REGION Network 71: Call CM Expel FWD/BWD (LBC_TwoWayActuator)
   RUNG wire#powerrail
      #instcmExpelFwdBwd(enable := wire#w1, enableManualCmds := wire#w2, parentReferenceDesignator := "Unit1.Em1.Config".em.referenceDesignator.combined, feedbackHomePos := "BA010AZCRBK01.01", feedbackWorkPos := "BA010AZCRBK01.11", interlockHomePos := "Unit1.Em1.ControlNodes".cm.interlock.expel.home, interlockWorkPos := "Unit1.Em1.ControlNodes".cm.interlock.expel.work, configuration := "Unit1.Em1.Config".cmExpelFwdBwd, moduleInterface := "Unit1.Em1.HmiInterface".cmExpelFwdBwd, controlNode := "Unit1.Em1.ControlNodes".cmExpelFwdBwd, goToHomePos => "BA010AZCRPM06.01", goToWorkPos => "BA010AZCRPM06.00")
   END_RUNG
   RUNG wire#powerrail
      I_Contact( #statUnitStatus.state.aborted )
   END_RUNG wire#w1
   RUNG wire#powerrail
      Contact( #statEnableManualCmds )
   END_RUNG wire#w2
   RUNG wire#powerrail
      Contact( #statRcEnableCmds )
   END_RUNG wire#w2
   // the same network as SCL:
   #instcmExpelFwdBwd(enable := NOT #statUnitStatus.state.aborted,   // "LBC_TwoWayActuatorCn"
                      parentReferenceDesignator := "Unit1.Em1.Config".em.referenceDesignator.combined,
                      feedbackHomePos := "BA010AZCRBK01.01",
                      feedbackWorkPos := "BA010AZCRBK01.11",
                      enableManualCmds := #statEnableManualCmds OR #statRcEnableCmds,
                      interlockHomePos := "Unit1.Em1.ControlNodes".cm.interlock.expel.home,
                      interlockWorkPos := "Unit1.Em1.ControlNodes".cm.interlock.expel.work,
                      configuration := "Unit1.Em1.Config".cmExpelFwdBwd,
                      moduleInterface := "Unit1.Em1.HmiInterface".cmExpelFwdBwd,
                      controlNode := "Unit1.Em1.ControlNodes".cmExpelFwdBwd,
                      goToHomePos => "BA010AZCRPM06.01",
                      goToWorkPos => "BA010AZCRPM06.00");
END_REGION

REGION Network 72: ******************** Control Modules (Accessories) ********************
END_REGION

REGION Network 73: Reset CMS
   RUNG wire#powerrail
      Contact( #statUnitStatus.acknowledgeActive )
      wire#w1
      Contact( "Unit1.Em1.ControlNodes".cmEpc.monitoring.error )
      Coil( "Unit1.Em1.ControlNodes".cmEpc.commands.reset )
   END_RUNG
   RUNG wire#powerrail
      Contact( #statUnitStatus.state.resetting )
   END_RUNG wire#w1
   RUNG wire#w1
      Contact( "Unit1.Em1.HmiInterface".cmBobinID.monitoring.error )
      Coil( "Unit1.Em1.HmiInterface".cmBobinID.commands.ResetReq )
   END_RUNG
   // the same network as SCL:
   #_w1 := #statUnitStatus.acknowledgeActive OR #statUnitStatus.state.resetting;
   "Unit1.Em1.ControlNodes".cmEpc.commands.reset := #_w1 AND "Unit1.Em1.ControlNodes".cmEpc.monitoring.error;
   "Unit1.Em1.HmiInterface".cmBobinID.commands.ResetReq := #_w1 AND "Unit1.Em1.HmiInterface".cmBobinID.monitoring.error;
END_REGION

REGION Network 74: Call CM EPC Commands
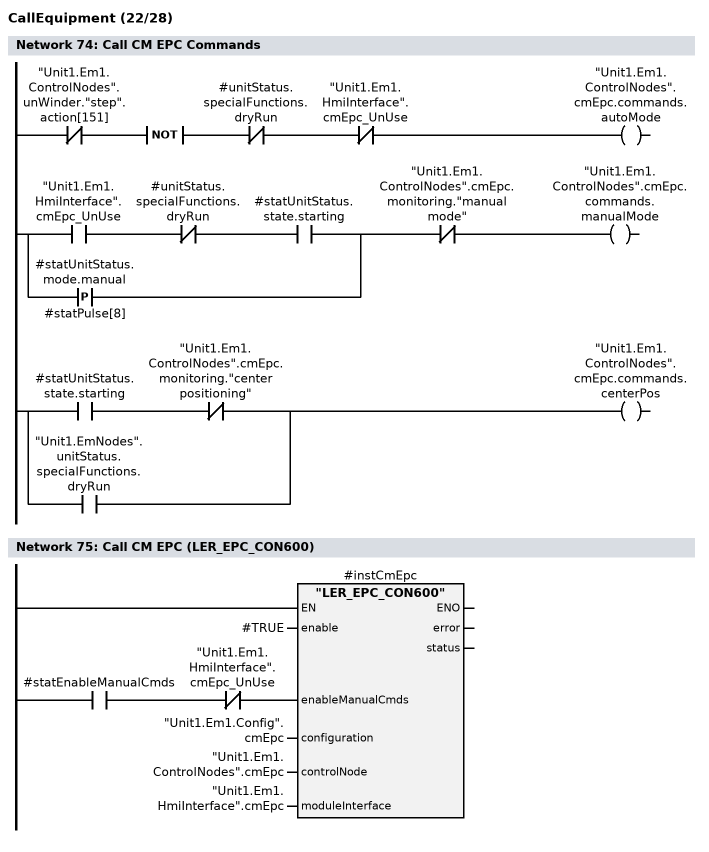
   RUNG wire#powerrail
      I_Contact( "Unit1.Em1.ControlNodes".unWinder."step".action[151] )
      Not()
      I_Contact( #unitStatus.specialFunctions.dryRun )
      I_Contact( "Unit1.Em1.HmiInterface".cmEpc_UnUse )
      Coil( "Unit1.Em1.ControlNodes".cmEpc.commands.autoMode )
   END_RUNG
   RUNG wire#powerrail
      Contact( "Unit1.Em1.HmiInterface".cmEpc_UnUse )
      I_Contact( #unitStatus.specialFunctions.dryRun )
      Contact( #statUnitStatus.state.starting )
      wire#w1
      I_Contact( "Unit1.Em1.ControlNodes".cmEpc.monitoring."manual mode" )
      Coil( "Unit1.Em1.ControlNodes".cmEpc.commands.manualMode )
   END_RUNG
   RUNG wire#powerrail
      P_Contact(operand := #statUnitStatus.mode.manual, bit := #statPulse[8])
   END_RUNG wire#w1
   RUNG wire#powerrail
      Contact( #statUnitStatus.state.starting )
      I_Contact( "Unit1.Em1.ControlNodes".cmEpc.monitoring."center positioning" )
      wire#w2
      Coil( "Unit1.Em1.ControlNodes".cmEpc.commands.centerPos )
   END_RUNG
   RUNG wire#powerrail
      Contact( "Unit1.EmNodes".unitStatus.specialFunctions.dryRun )
   END_RUNG wire#w2
   // the same network as SCL:
   "Unit1.Em1.ControlNodes".cmEpc.commands.autoMode := NOT (NOT "Unit1.Em1.ControlNodes".unWinder."step".action[151]) AND NOT #unitStatus.specialFunctions.dryRun AND NOT "Unit1.Em1.HmiInterface".cmEpc_UnUse;
   #_w1 := #statUnitStatus.mode.manual AND NOT #statPulse[8];   // rising edge of #statUnitStatus.mode.manual
   #statPulse[8] := #statUnitStatus.mode.manual;
   "Unit1.Em1.ControlNodes".cmEpc.commands.manualMode := (("Unit1.Em1.HmiInterface".cmEpc_UnUse AND NOT #unitStatus.specialFunctions.dryRun AND #statUnitStatus.state.starting) OR #_w1) AND NOT "Unit1.Em1.ControlNodes".cmEpc.monitoring."manual mode";
   "Unit1.Em1.ControlNodes".cmEpc.commands.centerPos := (#statUnitStatus.state.starting AND NOT "Unit1.Em1.ControlNodes".cmEpc.monitoring."center positioning") OR "Unit1.EmNodes".unitStatus.specialFunctions.dryRun;
END_REGION

REGION Network 75: Call CM EPC (LER_EPC_CON600)
   RUNG wire#powerrail
      #instCmEpc(enableManualCmds := wire#w1, enable := #TRUE, configuration := "Unit1.Em1.Config".cmEpc, controlNode := "Unit1.Em1.ControlNodes".cmEpc, moduleInterface := "Unit1.Em1.HmiInterface".cmEpc, error =>, status =>)
   END_RUNG
   RUNG wire#powerrail
      Contact( #statEnableManualCmds )
      I_Contact( "Unit1.Em1.HmiInterface".cmEpc_UnUse )
   END_RUNG wire#w1
   // the same network as SCL:
   #instCmEpc(enable := #TRUE,   // "LER_EPC_CON600"
              enableManualCmds := #statEnableManualCmds AND NOT "Unit1.Em1.HmiInterface".cmEpc_UnUse,
              configuration := "Unit1.Em1.Config".cmEpc,
              controlNode := "Unit1.Em1.ControlNodes".cmEpc,
              moduleInterface := "Unit1.Em1.HmiInterface".cmEpc);
END_REGION

REGION Network 76: ******************** Feedback to Unit ********************
END_REGION

REGION Network 77: Determine StateComplete (SC) in Mode Production
   // Conditions for the Equipment Modules "stateComplete" feedback to the unit. This feedback is given when the task in for the respective state is complete.
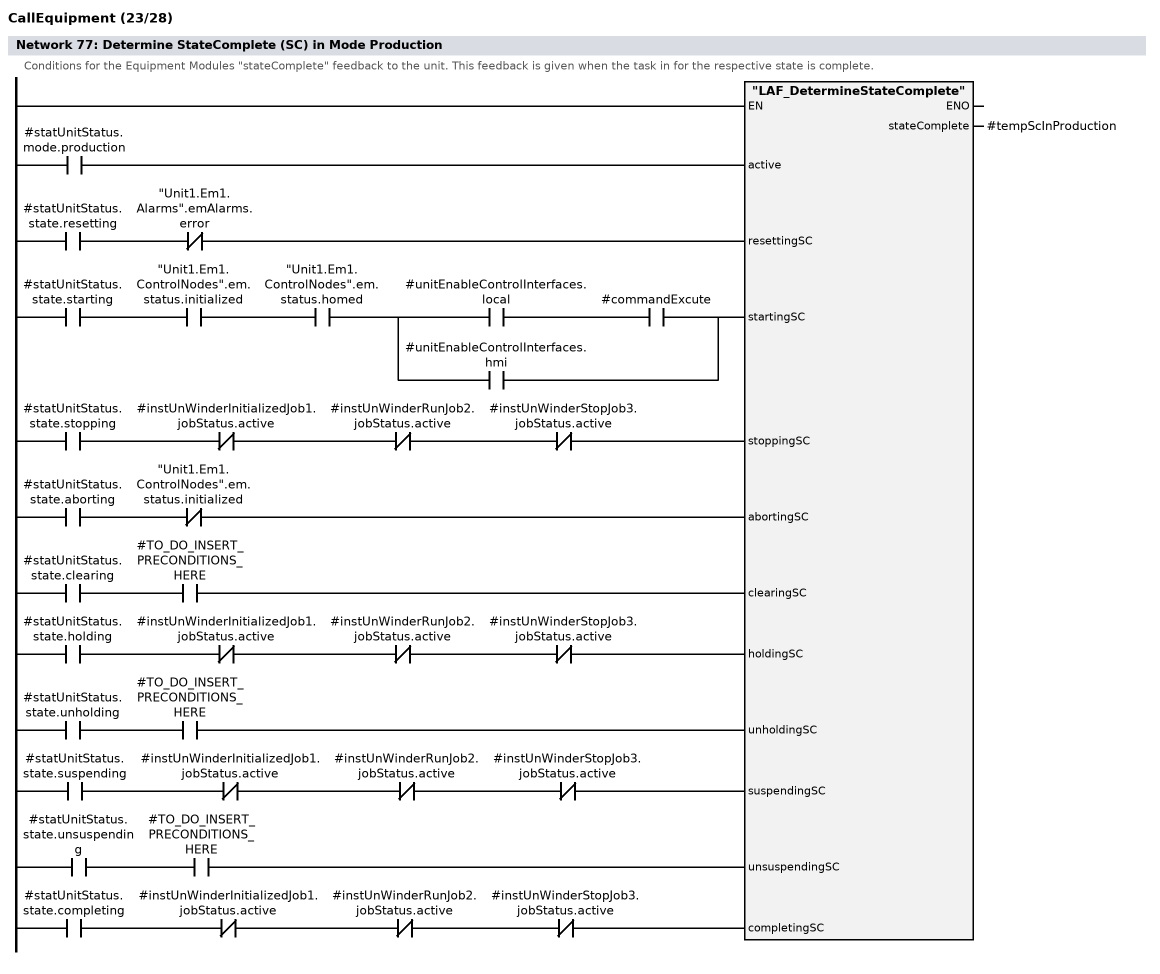
   RUNG wire#powerrail
      "LAF_DetermineStateComplete"(active := wire#w1, resettingSC := wire#w2, startingSC := wire#w4, stoppingSC := wire#w5, abortingSC := wire#w6, clearingSC := wire#w7, holdingSC := wire#w8, unholdingSC := wire#w9, suspendingSC := wire#w10, unsuspendingSC := wire#w11, completingSC := wire#w12, stateComplete => #tempScInProduction)
   END_RUNG
   RUNG wire#powerrail
      Contact( #statUnitStatus.mode.production )
   END_RUNG wire#w1
   RUNG wire#powerrail
      Contact( #statUnitStatus.state.resetting )
      I_Contact( "Unit1.Em1.Alarms".emAlarms.error )
   END_RUNG wire#w2
   RUNG wire#powerrail
      Contact( #statUnitStatus.state.starting )
      Contact( "Unit1.Em1.ControlNodes".em.status.initialized )
      Contact( "Unit1.Em1.ControlNodes".em.status.homed )
      wire#w3
      Contact( #unitEnableControlInterfaces.local )
      Contact( #commandExcute )
   END_RUNG wire#w4
   RUNG wire#w3
      Contact( #unitEnableControlInterfaces.hmi )
   END_RUNG wire#w4
   RUNG wire#powerrail
      Contact( #statUnitStatus.state.stopping )
      I_Contact( #instUnWinderInitializedJob1.jobStatus.active )
      I_Contact( #instUnWinderRunJob2.jobStatus.active )
      I_Contact( #instUnWinderStopJob3.jobStatus.active )
   END_RUNG wire#w5
   RUNG wire#powerrail
      Contact( #statUnitStatus.state.aborting )
      I_Contact( "Unit1.Em1.ControlNodes".em.status.initialized )
   END_RUNG wire#w6
   RUNG wire#powerrail
      Contact( #statUnitStatus.state.clearing )
      Contact( #TO_DO_INSERT_PRECONDITIONS_HERE )
   END_RUNG wire#w7
   RUNG wire#powerrail
      Contact( #statUnitStatus.state.holding )
      I_Contact( #instUnWinderInitializedJob1.jobStatus.active )
      I_Contact( #instUnWinderRunJob2.jobStatus.active )
      I_Contact( #instUnWinderStopJob3.jobStatus.active )
   END_RUNG wire#w8
   RUNG wire#powerrail
      Contact( #statUnitStatus.state.unholding )
      Contact( #TO_DO_INSERT_PRECONDITIONS_HERE )
   END_RUNG wire#w9
   RUNG wire#powerrail
      Contact( #statUnitStatus.state.suspending )
      I_Contact( #instUnWinderInitializedJob1.jobStatus.active )
      I_Contact( #instUnWinderRunJob2.jobStatus.active )
      I_Contact( #instUnWinderStopJob3.jobStatus.active )
   END_RUNG wire#w10
   RUNG wire#powerrail
      Contact( #statUnitStatus.state.unsuspending )
      Contact( #TO_DO_INSERT_PRECONDITIONS_HERE )
   END_RUNG wire#w11
   RUNG wire#powerrail
      Contact( #statUnitStatus.state.completing )
      I_Contact( #instUnWinderInitializedJob1.jobStatus.active )
      I_Contact( #instUnWinderRunJob2.jobStatus.active )
      I_Contact( #instUnWinderStopJob3.jobStatus.active )
   END_RUNG wire#w12
   // the same network as SCL:
   "LAF_DetermineStateComplete"(active := #statUnitStatus.mode.production,
                           resettingSC := #statUnitStatus.state.resetting AND NOT "Unit1.Em1.Alarms".emAlarms.error,
                           startingSC := #statUnitStatus.state.starting AND "Unit1.Em1.ControlNodes".em.status.initialized AND "Unit1.Em1.ControlNodes".em.status.homed AND ((#unitEnableControlInterfaces.local AND #commandExcute) OR #unitEnableControlInterfaces.hmi),
                           stoppingSC := #statUnitStatus.state.stopping AND NOT #instUnWinderInitializedJob1.jobStatus.active AND NOT #instUnWinderRunJob2.jobStatus.active AND NOT #instUnWinderStopJob3.jobStatus.active,
                           abortingSC := #statUnitStatus.state.aborting AND NOT "Unit1.Em1.ControlNodes".em.status.initialized,
                           clearingSC := #statUnitStatus.state.clearing AND #TO_DO_INSERT_PRECONDITIONS_HERE,
                           holdingSC := #statUnitStatus.state.holding AND NOT #instUnWinderInitializedJob1.jobStatus.active AND NOT #instUnWinderRunJob2.jobStatus.active AND NOT #instUnWinderStopJob3.jobStatus.active,
                           unholdingSC := #statUnitStatus.state.unholding AND #TO_DO_INSERT_PRECONDITIONS_HERE,
                           suspendingSC := #statUnitStatus.state.suspending AND NOT #instUnWinderInitializedJob1.jobStatus.active AND NOT #instUnWinderRunJob2.jobStatus.active AND NOT #instUnWinderStopJob3.jobStatus.active,
                           unsuspendingSC := #statUnitStatus.state.unsuspending AND #TO_DO_INSERT_PRECONDITIONS_HERE,
                           completingSC := #statUnitStatus.state.completing AND NOT #instUnWinderInitializedJob1.jobStatus.active AND NOT #instUnWinderRunJob2.jobStatus.active AND NOT #instUnWinderStopJob3.jobStatus.active,
                           stateComplete => #tempScInProduction);
END_REGION

REGION Network 78: Determine StateComplete (SC) in Mode Maintenance/Manual
   // Conditions for the Equipment Modules "stateComplete" feedback to the unit. This feedback is given when the task in for the respective state is complete.
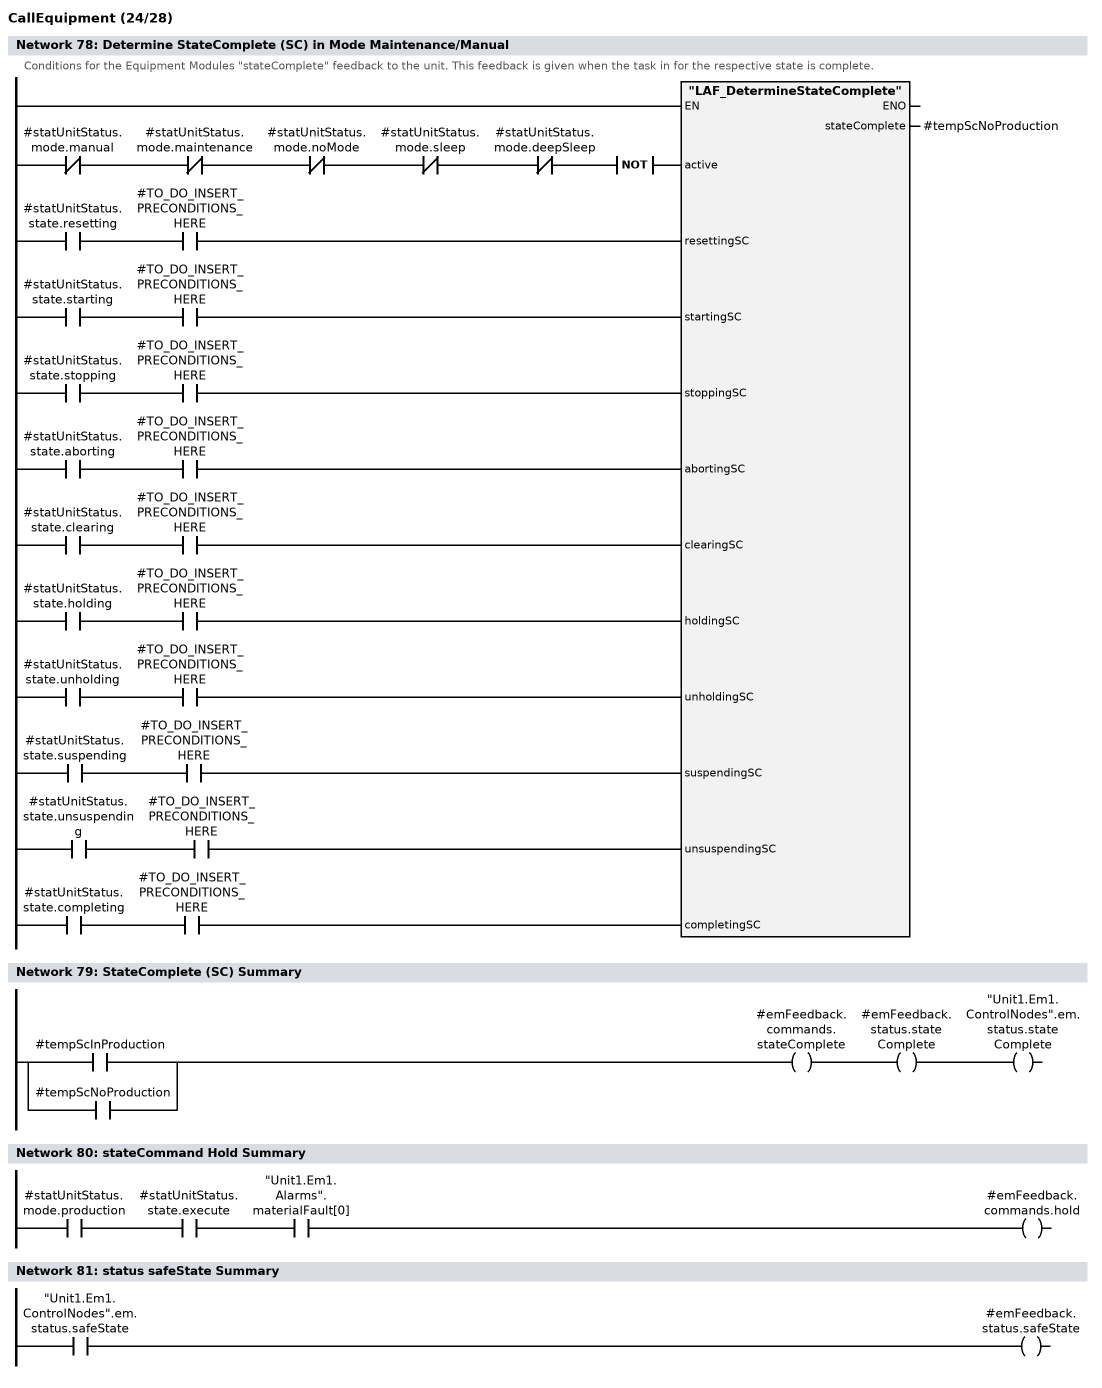
   RUNG wire#powerrail
      "LAF_DetermineStateComplete"(active := wire#w1, resettingSC := wire#w2, startingSC := wire#w3, stoppingSC := wire#w4, abortingSC := wire#w5, clearingSC := wire#w6, holdingSC := wire#w7, unholdingSC := wire#w8, suspendingSC := wire#w9, unsuspendingSC := wire#w10, completingSC := wire#w11, stateComplete => #tempScNoProduction)
   END_RUNG
   RUNG wire#powerrail
      I_Contact( #statUnitStatus.mode.manual )
      I_Contact( #statUnitStatus.mode.maintenance )
      I_Contact( #statUnitStatus.mode.noMode )
      I_Contact( #statUnitStatus.mode.sleep )
      I_Contact( #statUnitStatus.mode.deepSleep )
      Not()
   END_RUNG wire#w1
   RUNG wire#powerrail
      Contact( #statUnitStatus.state.resetting )
      Contact( #TO_DO_INSERT_PRECONDITIONS_HERE )
   END_RUNG wire#w2
   RUNG wire#powerrail
      Contact( #statUnitStatus.state.starting )
      Contact( #TO_DO_INSERT_PRECONDITIONS_HERE )
   END_RUNG wire#w3
   RUNG wire#powerrail
      Contact( #statUnitStatus.state.stopping )
      Contact( #TO_DO_INSERT_PRECONDITIONS_HERE )
   END_RUNG wire#w4
   RUNG wire#powerrail
      Contact( #statUnitStatus.state.aborting )
      Contact( #TO_DO_INSERT_PRECONDITIONS_HERE )
   END_RUNG wire#w5
   RUNG wire#powerrail
      Contact( #statUnitStatus.state.clearing )
      Contact( #TO_DO_INSERT_PRECONDITIONS_HERE )
   END_RUNG wire#w6
   RUNG wire#powerrail
      Contact( #statUnitStatus.state.holding )
      Contact( #TO_DO_INSERT_PRECONDITIONS_HERE )
   END_RUNG wire#w7
   RUNG wire#powerrail
      Contact( #statUnitStatus.state.unholding )
      Contact( #TO_DO_INSERT_PRECONDITIONS_HERE )
   END_RUNG wire#w8
   RUNG wire#powerrail
      Contact( #statUnitStatus.state.suspending )
      Contact( #TO_DO_INSERT_PRECONDITIONS_HERE )
   END_RUNG wire#w9
   RUNG wire#powerrail
      Contact( #statUnitStatus.state.unsuspending )
      Contact( #TO_DO_INSERT_PRECONDITIONS_HERE )
   END_RUNG wire#w10
   RUNG wire#powerrail
      Contact( #statUnitStatus.state.completing )
      Contact( #TO_DO_INSERT_PRECONDITIONS_HERE )
   END_RUNG wire#w11
   // the same network as SCL:
   "LAF_DetermineStateComplete"(active := NOT (NOT #statUnitStatus.mode.manual AND NOT #statUnitStatus.mode.maintenance AND NOT #statUnitStatus.mode.noMode AND NOT #statUnitStatus.mode.sleep AND NOT #statUnitStatus.mode.deepSleep),
                           resettingSC := #statUnitStatus.state.resetting AND #TO_DO_INSERT_PRECONDITIONS_HERE,
                           startingSC := #statUnitStatus.state.starting AND #TO_DO_INSERT_PRECONDITIONS_HERE,
                           stoppingSC := #statUnitStatus.state.stopping AND #TO_DO_INSERT_PRECONDITIONS_HERE,
                           abortingSC := #statUnitStatus.state.aborting AND #TO_DO_INSERT_PRECONDITIONS_HERE,
                           clearingSC := #statUnitStatus.state.clearing AND #TO_DO_INSERT_PRECONDITIONS_HERE,
                           holdingSC := #statUnitStatus.state.holding AND #TO_DO_INSERT_PRECONDITIONS_HERE,
                           unholdingSC := #statUnitStatus.state.unholding AND #TO_DO_INSERT_PRECONDITIONS_HERE,
                           suspendingSC := #statUnitStatus.state.suspending AND #TO_DO_INSERT_PRECONDITIONS_HERE,
                           unsuspendingSC := #statUnitStatus.state.unsuspending AND #TO_DO_INSERT_PRECONDITIONS_HERE,
                           completingSC := #statUnitStatus.state.completing AND #TO_DO_INSERT_PRECONDITIONS_HERE,
                           stateComplete => #tempScNoProduction);
END_REGION

REGION Network 79: StateComplete (SC) Summary
   RUNG wire#powerrail
      Contact( #tempScInProduction )
      wire#w1
      Coil( #emFeedback.commands.stateComplete )
      Coil( #emFeedback.status.stateComplete )
      Coil( "Unit1.Em1.ControlNodes".em.status.stateComplete )
   END_RUNG
   RUNG wire#powerrail
      Contact( #tempScNoProduction )
   END_RUNG wire#w1
   // the same network as SCL:
   #emFeedback.commands.stateComplete := #tempScInProduction OR #tempScNoProduction;
   #emFeedback.status.stateComplete := #emFeedback.commands.stateComplete;
   "Unit1.Em1.ControlNodes".em.status.stateComplete := #emFeedback.commands.stateComplete;
END_REGION

REGION Network 80: stateCommand Hold Summary
   RUNG wire#powerrail
      Contact( #statUnitStatus.mode.production )
      Contact( #statUnitStatus.state.execute )
      Contact( "Unit1.Em1.Alarms".materialFault[0] )
      Coil( #emFeedback.commands.hold )
   END_RUNG
   // the same network as SCL:
   #emFeedback.commands.hold := #statUnitStatus.mode.production AND #statUnitStatus.state.execute AND "Unit1.Em1.Alarms".materialFault[0];
END_REGION

REGION Network 81: status safeState Summary
   RUNG wire#powerrail
      Contact( "Unit1.Em1.ControlNodes".em.status.safeState )
      Coil( #emFeedback.status.safeState )
   END_RUNG
   // the same network as SCL:
   #emFeedback.status.safeState := "Unit1.Em1.ControlNodes".em.status.safeState;
END_REGION

REGION Network 82: status safetyReleased Summary
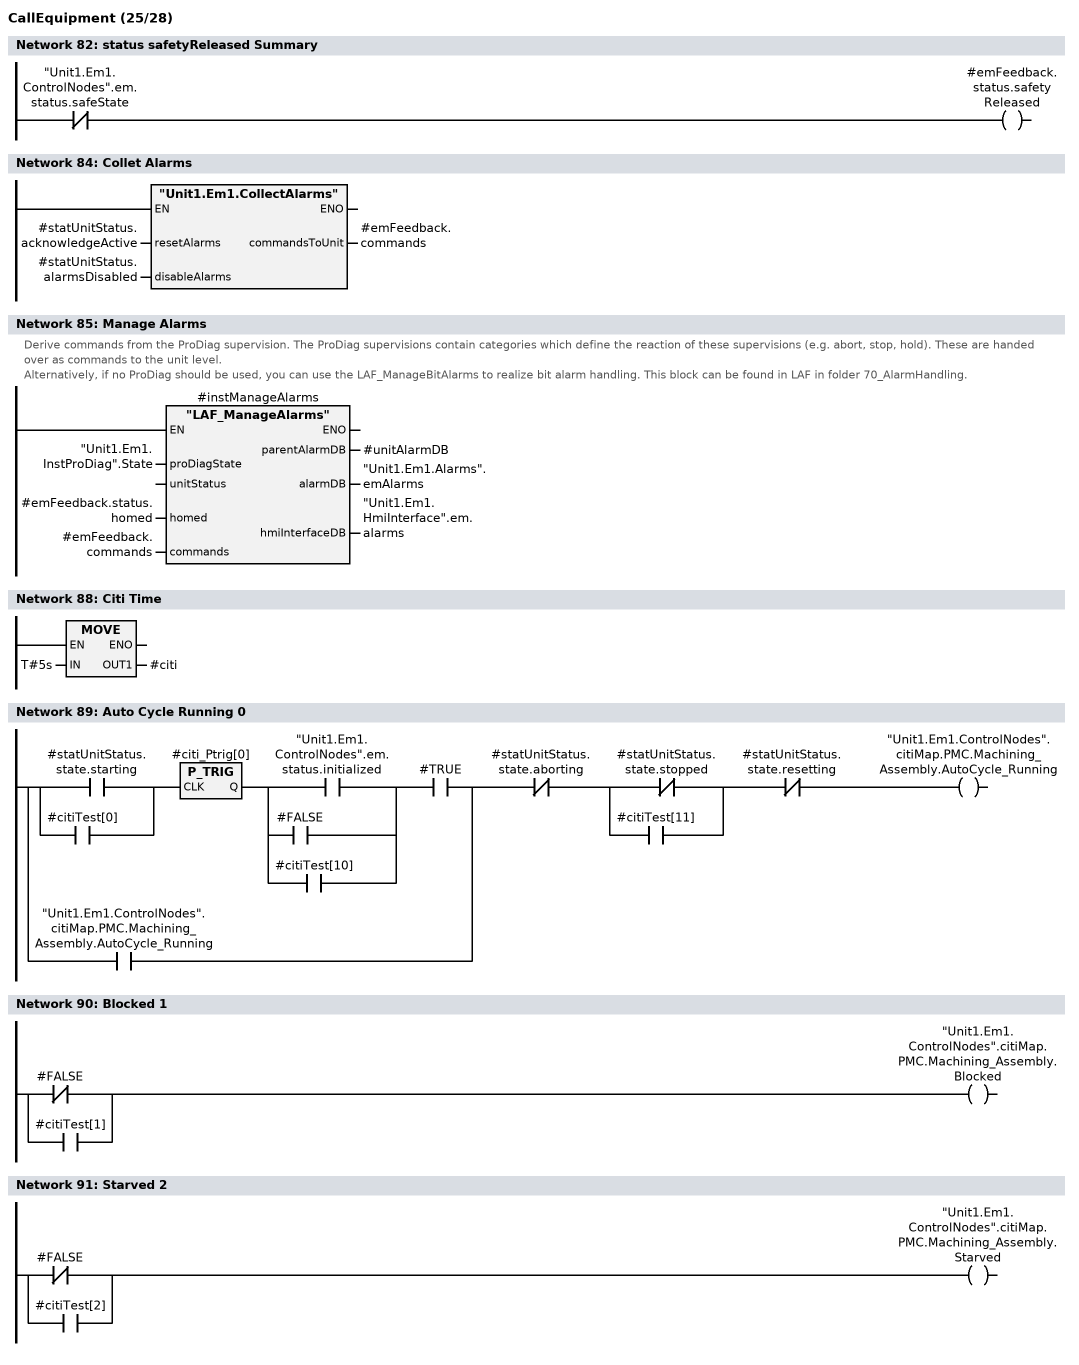
   RUNG wire#powerrail
      I_Contact( "Unit1.Em1.ControlNodes".em.status.safeState )
      Coil( #emFeedback.status.safetyReleased )
   END_RUNG
   // the same network as SCL:
   #emFeedback.status.safetyReleased := NOT "Unit1.Em1.ControlNodes".em.status.safeState;
END_REGION

REGION Network 83: ******************** Alarms ********************
END_REGION

REGION Network 84: Collet Alarms
   RUNG wire#powerrail
      "Unit1.Em1.CollectAlarms"(resetAlarms := #statUnitStatus.acknowledgeActive, disableAlarms := #statUnitStatus.alarmsDisabled, commandsToUnit => #emFeedback.commands)
   END_RUNG
   // the same network as SCL:
   "Unit1.Em1.CollectAlarms"(resetAlarms := #statUnitStatus.acknowledgeActive,
                           disableAlarms := #statUnitStatus.alarmsDisabled,
                           commandsToUnit => #emFeedback.commands);
END_REGION

REGION Network 85: Manage Alarms
   // Derive commands from the ProDiag supervision. The ProDiag supervisions contain categories which define the reaction of these supervisions (e.g. abort, stop, hold). These are handed over as commands to the unit level.
   // Alternatively, if no ProDiag should be used, you can use the LAF_ManageBitAlarms to realize bit alarm handling. This block can be found in LAF in folder 70_AlarmHandling.
   RUNG wire#powerrail
      #instManageAlarms(proDiagState := "Unit1.Em1.InstProDiag".State, unitStatus :=, homed := #emFeedback.status.homed, commands := #emFeedback.commands, parentAlarmDB => #unitAlarmDB, alarmDB => "Unit1.Em1.Alarms".emAlarms, hmiInterfaceDB => "Unit1.Em1.HmiInterface".em.alarms)
   END_RUNG
   // the same network as SCL:
   #instManageAlarms(proDiagState := "Unit1.Em1.InstProDiag".State,   // "LAF_ManageAlarms"
                     homed := #emFeedback.status.homed,
                     commands := #emFeedback.commands,
                     parentAlarmDB => #unitAlarmDB,
                     alarmDB => "Unit1.Em1.Alarms".emAlarms,
                     hmiInterfaceDB => "Unit1.Em1.HmiInterface".em.alarms);
END_REGION

REGION Network 87: ******************** CITI ********************
END_REGION

REGION Network 88: Citi Time
   RUNG wire#powerrail
      Move(in := T#5s, out1 => #citi)
   END_RUNG
   // the same network as SCL:
   #citi := T#5s;
END_REGION

REGION Network 89: Auto Cycle Running 0
   RUNG wire#powerrail
      Contact( #statUnitStatus.state.starting )
      wire#w1
      P_Trig( #citi_Ptrig[0] )
      wire#w2
      Contact( "Unit1.Em1.ControlNodes".em.status.initialized )
      wire#w3
      Contact( #TRUE )
      wire#w4
      I_Contact( #statUnitStatus.state.aborting )
      wire#w5
      I_Contact( #statUnitStatus.state.stopped )
      wire#w6
      I_Contact( #statUnitStatus.state.resetting )
      Coil( "Unit1.Em1.ControlNodes".citiMap.PMC.Machining_Assembly.AutoCycle_Running )
   END_RUNG
   RUNG wire#powerrail
      Contact( #citiTest[0] )
   END_RUNG wire#w1
   RUNG wire#w2
      Contact( #FALSE )
   END_RUNG wire#w3
   RUNG wire#w2
      Contact( #citiTest[10] )
   END_RUNG wire#w3
   RUNG wire#powerrail
      Contact( "Unit1.Em1.ControlNodes".citiMap.PMC.Machining_Assembly.AutoCycle_Running )
   END_RUNG wire#w4
   RUNG wire#w5
      Contact( #citiTest[11] )
   END_RUNG wire#w6
   // the same network as SCL:
   #_w1 := #statUnitStatus.state.starting OR #citiTest[0];
   #_w2 := #_w1 AND NOT #citi_Ptrig[0];   // rising edge
   #citi_Ptrig[0] := #_w1;
   "Unit1.Em1.ControlNodes".citiMap.PMC.Machining_Assembly.AutoCycle_Running := ((#_w2 AND ("Unit1.Em1.ControlNodes".em.status.initialized OR #FALSE OR #citiTest[10]) AND #TRUE) OR "Unit1.Em1.ControlNodes".citiMap.PMC.Machining_Assembly.AutoCycle_Running) AND NOT #statUnitStatus.state.aborting AND (NOT #statUnitStatus.state.stopped OR #citiTest[11]) AND NOT #statUnitStatus.state.resetting;
END_REGION

REGION Network 90: Blocked 1
   RUNG wire#powerrail
      I_Contact( #FALSE )
      wire#w1
      Coil( "Unit1.Em1.ControlNodes".citiMap.PMC.Machining_Assembly.Blocked )
   END_RUNG
   RUNG wire#powerrail
      Contact( #citiTest[1] )
   END_RUNG wire#w1
   // the same network as SCL:
   "Unit1.Em1.ControlNodes".citiMap.PMC.Machining_Assembly.Blocked := NOT #FALSE OR #citiTest[1];
END_REGION

REGION Network 91: Starved 2
   RUNG wire#powerrail
      I_Contact( #FALSE )
      wire#w1
      Coil( "Unit1.Em1.ControlNodes".citiMap.PMC.Machining_Assembly.Starved )
   END_RUNG
   RUNG wire#powerrail
      Contact( #citiTest[2] )
   END_RUNG wire#w1
   // the same network as SCL:
   "Unit1.Em1.ControlNodes".citiMap.PMC.Machining_Assembly.Starved := NOT #FALSE OR #citiTest[2];
END_REGION

REGION Network 92: Good Count 3
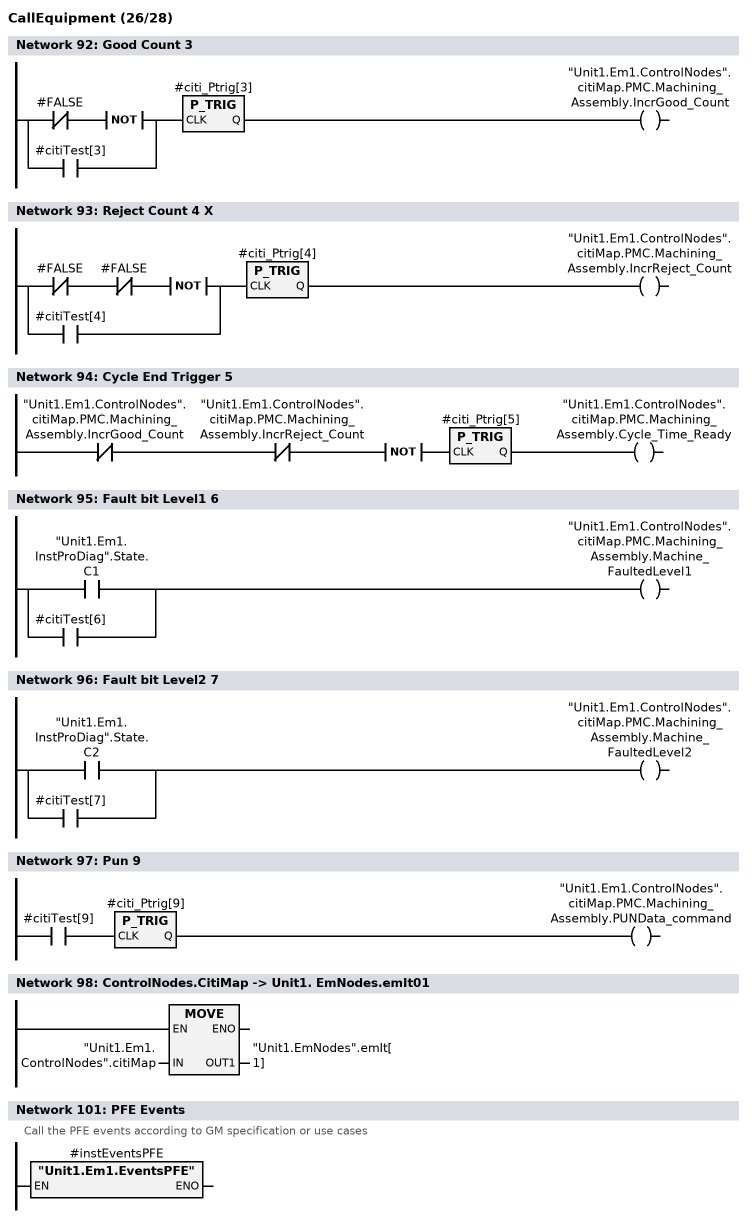
   RUNG wire#powerrail
      I_Contact( #FALSE )
      Not()
      wire#w1
      P_Trig( #citi_Ptrig[3] )
      Coil( "Unit1.Em1.ControlNodes".citiMap.PMC.Machining_Assembly.IncrGood_Count )
   END_RUNG
   RUNG wire#powerrail
      Contact( #citiTest[3] )
   END_RUNG wire#w1
   // the same network as SCL:
   #_w1 := NOT (NOT #FALSE) OR #citiTest[3];
   #_w2 := #_w1 AND NOT #citi_Ptrig[3];   // rising edge
   #citi_Ptrig[3] := #_w1;
   "Unit1.Em1.ControlNodes".citiMap.PMC.Machining_Assembly.IncrGood_Count := #_w2;
END_REGION

REGION Network 93: Reject Count 4 X
   RUNG wire#powerrail
      I_Contact( #FALSE )
      I_Contact( #FALSE )
      Not()
      wire#w1
      P_Trig( #citi_Ptrig[4] )
      Coil( "Unit1.Em1.ControlNodes".citiMap.PMC.Machining_Assembly.IncrReject_Count )
   END_RUNG
   RUNG wire#powerrail
      Contact( #citiTest[4] )
   END_RUNG wire#w1
   // the same network as SCL:
   #_w1 := NOT (NOT #FALSE AND NOT #FALSE) OR #citiTest[4];
   #_w2 := #_w1 AND NOT #citi_Ptrig[4];   // rising edge
   #citi_Ptrig[4] := #_w1;
   "Unit1.Em1.ControlNodes".citiMap.PMC.Machining_Assembly.IncrReject_Count := #_w2;
END_REGION

REGION Network 94: Cycle End Trigger 5
   RUNG wire#powerrail
      I_Contact( "Unit1.Em1.ControlNodes".citiMap.PMC.Machining_Assembly.IncrGood_Count )
      I_Contact( "Unit1.Em1.ControlNodes".citiMap.PMC.Machining_Assembly.IncrReject_Count )
      Not()
      P_Trig( #citi_Ptrig[5] )
      Coil( "Unit1.Em1.ControlNodes".citiMap.PMC.Machining_Assembly.Cycle_Time_Ready )
   END_RUNG
   // the same network as SCL:
   #_w1 := NOT (NOT "Unit1.Em1.ControlNodes".citiMap.PMC.Machining_Assembly.IncrGood_Count AND NOT "Unit1.Em1.ControlNodes".citiMap.PMC.Machining_Assembly.IncrReject_Count);
   #_w2 := #_w1 AND NOT #citi_Ptrig[5];   // rising edge
   #citi_Ptrig[5] := #_w1;
   "Unit1.Em1.ControlNodes".citiMap.PMC.Machining_Assembly.Cycle_Time_Ready := #_w2;
END_REGION

REGION Network 95: Fault bit Level1 6
   RUNG wire#powerrail
      Contact( "Unit1.Em1.InstProDiag".State.C1 )
      wire#w1
      Coil( "Unit1.Em1.ControlNodes".citiMap.PMC.Machining_Assembly.Machine_FaultedLevel1 )
   END_RUNG
   RUNG wire#powerrail
      Contact( #citiTest[6] )
   END_RUNG wire#w1
   // the same network as SCL:
   "Unit1.Em1.ControlNodes".citiMap.PMC.Machining_Assembly.Machine_FaultedLevel1 := "Unit1.Em1.InstProDiag".State.C1 OR #citiTest[6];
END_REGION

REGION Network 96: Fault bit Level2 7
   RUNG wire#powerrail
      Contact( "Unit1.Em1.InstProDiag".State.C2 )
      wire#w1
      Coil( "Unit1.Em1.ControlNodes".citiMap.PMC.Machining_Assembly.Machine_FaultedLevel2 )
   END_RUNG
   RUNG wire#powerrail
      Contact( #citiTest[7] )
   END_RUNG wire#w1
   // the same network as SCL:
   "Unit1.Em1.ControlNodes".citiMap.PMC.Machining_Assembly.Machine_FaultedLevel2 := "Unit1.Em1.InstProDiag".State.C2 OR #citiTest[7];
END_REGION

REGION Network 97: Pun 9
   RUNG wire#powerrail
      Contact( #citiTest[9] )
      P_Trig( #citi_Ptrig[9] )
      Coil( "Unit1.Em1.ControlNodes".citiMap.PMC.Machining_Assembly.PUNData_command )
   END_RUNG
   // the same network as SCL:
   #_w1 := #citiTest[9] AND NOT #citi_Ptrig[9];   // rising edge
   #citi_Ptrig[9] := #citiTest[9];
   "Unit1.Em1.ControlNodes".citiMap.PMC.Machining_Assembly.PUNData_command := #_w1;
END_REGION

REGION Network 98: ControlNodes.CitiMap -> Unit1. EmNodes.emIt01
   RUNG wire#powerrail
      Move(in := "Unit1.Em1.ControlNodes".citiMap, out1 => "Unit1.EmNodes".emIt[1])
   END_RUNG
   // the same network as SCL:
   "Unit1.EmNodes".emIt[1] := "Unit1.Em1.ControlNodes".citiMap;
END_REGION

REGION Network 100: ******************** PFE Events ********************
END_REGION

REGION Network 101: PFE Events
   // Call the PFE events according to GM specification or use cases
   RUNG wire#powerrail
      #instEventsPFE()
   END_RUNG
   // the same network as SCL:
   #instEventsPFE();   // "Unit1.Em1.EventsPFE"
END_REGION

REGION Network 102: ******************** EM Relations Output ********************
END_REGION

REGION Network 103: EM1 Job Interface
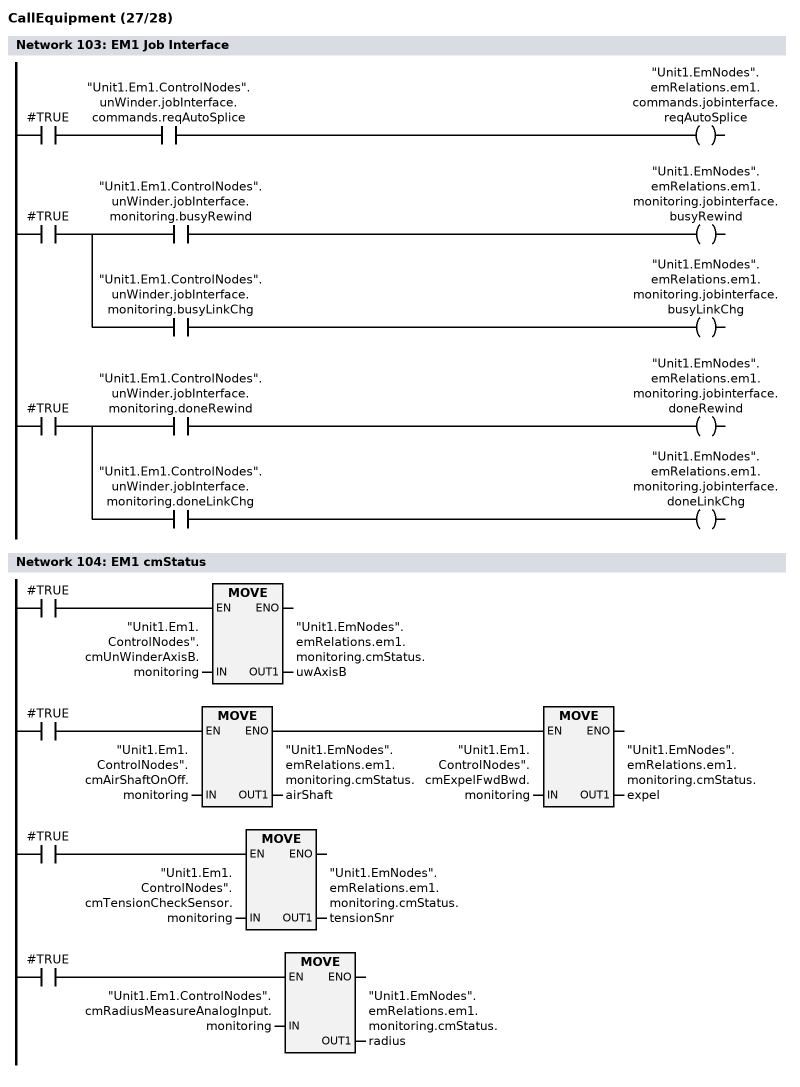
   RUNG wire#powerrail
      Contact( #TRUE )
      Contact( "Unit1.Em1.ControlNodes".unWinder.jobInterface.commands.reqAutoSplice )
      Coil( "Unit1.EmNodes".emRelations.em1.commands.jobinterface.reqAutoSplice )
   END_RUNG
   RUNG wire#powerrail
      Contact( #TRUE )
      wire#w1
      Contact( "Unit1.Em1.ControlNodes".unWinder.jobInterface.monitoring.busyRewind )
      Coil( "Unit1.EmNodes".emRelations.em1.monitoring.jobinterface.busyRewind )
   END_RUNG
   RUNG wire#w1
      Contact( "Unit1.Em1.ControlNodes".unWinder.jobInterface.monitoring.busyLinkChg )
      Coil( "Unit1.EmNodes".emRelations.em1.monitoring.jobinterface.busyLinkChg )
   END_RUNG
   RUNG wire#powerrail
      Contact( #TRUE )
      wire#w2
      Contact( "Unit1.Em1.ControlNodes".unWinder.jobInterface.monitoring.doneRewind )
      Coil( "Unit1.EmNodes".emRelations.em1.monitoring.jobinterface.doneRewind )
   END_RUNG
   RUNG wire#w2
      Contact( "Unit1.Em1.ControlNodes".unWinder.jobInterface.monitoring.doneLinkChg )
      Coil( "Unit1.EmNodes".emRelations.em1.monitoring.jobinterface.doneLinkChg )
   END_RUNG
   // the same network as SCL:
   "Unit1.EmNodes".emRelations.em1.commands.jobinterface.reqAutoSplice := #TRUE AND "Unit1.Em1.ControlNodes".unWinder.jobInterface.commands.reqAutoSplice;
   "Unit1.EmNodes".emRelations.em1.monitoring.jobinterface.busyRewind := #TRUE AND "Unit1.Em1.ControlNodes".unWinder.jobInterface.monitoring.busyRewind;
   "Unit1.EmNodes".emRelations.em1.monitoring.jobinterface.busyLinkChg := #TRUE AND "Unit1.Em1.ControlNodes".unWinder.jobInterface.monitoring.busyLinkChg;
   "Unit1.EmNodes".emRelations.em1.monitoring.jobinterface.doneRewind := #TRUE AND "Unit1.Em1.ControlNodes".unWinder.jobInterface.monitoring.doneRewind;
   "Unit1.EmNodes".emRelations.em1.monitoring.jobinterface.doneLinkChg := #TRUE AND "Unit1.Em1.ControlNodes".unWinder.jobInterface.monitoring.doneLinkChg;
END_REGION

REGION Network 104: EM1 cmStatus
   RUNG wire#powerrail
      Contact( #TRUE )
      Move(in := "Unit1.Em1.ControlNodes".cmUnWinderAxisB.monitoring, out1 => "Unit1.EmNodes".emRelations.em1.monitoring.cmStatus.uwAxisB)
   END_RUNG
   RUNG wire#powerrail
      Contact( #TRUE )
      Move(in := "Unit1.Em1.ControlNodes".cmAirShaftOnOff.monitoring, out1 => "Unit1.EmNodes".emRelations.em1.monitoring.cmStatus.airShaft)
      Move(in := "Unit1.Em1.ControlNodes".cmExpelFwdBwd.monitoring, out1 => "Unit1.EmNodes".emRelations.em1.monitoring.cmStatus.expel)
   END_RUNG
   RUNG wire#powerrail
      Contact( #TRUE )
      Move(in := "Unit1.Em1.ControlNodes".cmTensionCheckSensor.monitoring, out1 => "Unit1.EmNodes".emRelations.em1.monitoring.cmStatus.tensionSnr)
   END_RUNG
   RUNG wire#powerrail
      Contact( #TRUE )
      Move(in := "Unit1.Em1.ControlNodes".cmRadiusMeasureAnalogInput.monitoring, out1 => "Unit1.EmNodes".emRelations.em1.monitoring.cmStatus.radius)
   END_RUNG
   // the same network as SCL:
   IF #TRUE THEN
       "Unit1.EmNodes".emRelations.em1.monitoring.cmStatus.uwAxisB := "Unit1.Em1.ControlNodes".cmUnWinderAxisB.monitoring;
       "Unit1.EmNodes".emRelations.em1.monitoring.cmStatus.airShaft := "Unit1.Em1.ControlNodes".cmAirShaftOnOff.monitoring;
       "Unit1.EmNodes".emRelations.em1.monitoring.cmStatus.expel := "Unit1.Em1.ControlNodes".cmExpelFwdBwd.monitoring;
       "Unit1.EmNodes".emRelations.em1.monitoring.cmStatus.tensionSnr := "Unit1.Em1.ControlNodes".cmTensionCheckSensor.monitoring;
       "Unit1.EmNodes".emRelations.em1.monitoring.cmStatus.radius := "Unit1.Em1.ControlNodes".cmRadiusMeasureAnalogInput.monitoring;
   END_IF;
END_REGION

REGION Network 105: EM1 UserDefine
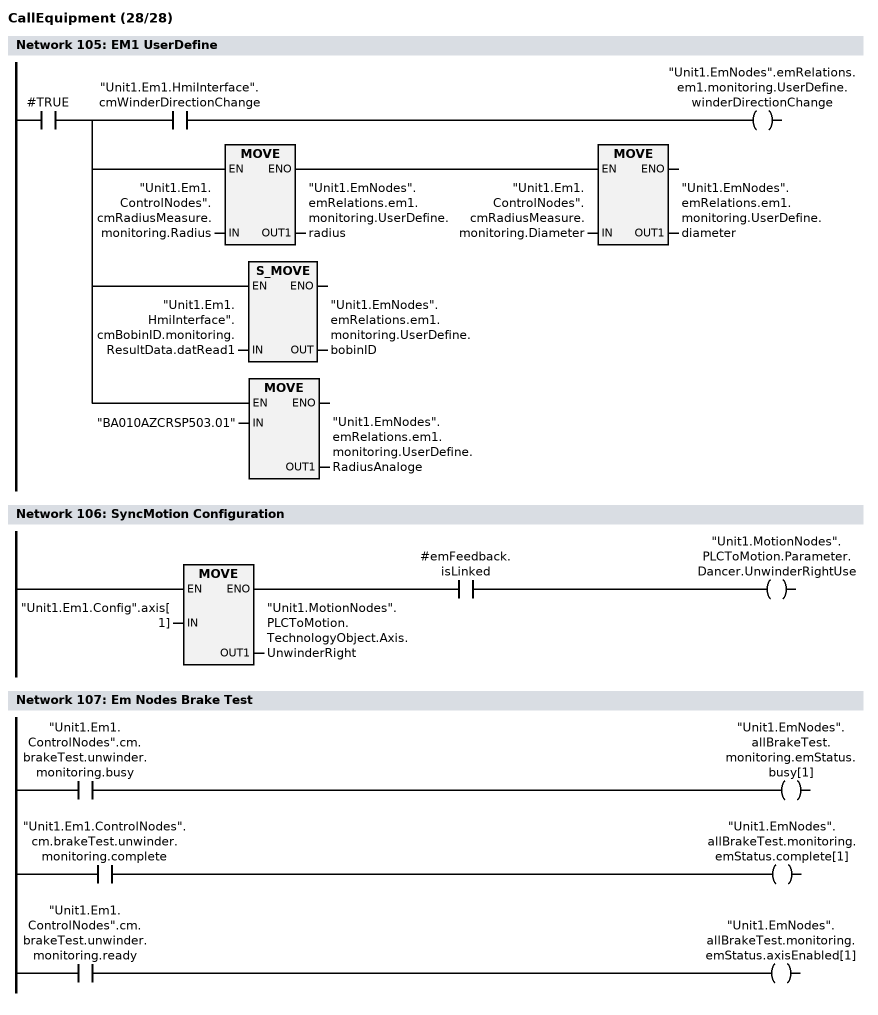
   RUNG wire#powerrail
      Contact( #TRUE )
      wire#w1
      Contact( "Unit1.Em1.HmiInterface".cmWinderDirectionChange )
      Coil( "Unit1.EmNodes".emRelations.em1.monitoring.UserDefine.winderDirectionChange )
   END_RUNG
   RUNG wire#w1
      Move(in := "Unit1.Em1.ControlNodes".cmRadiusMeasure.monitoring.Radius, out1 => "Unit1.EmNodes".emRelations.em1.monitoring.UserDefine.radius)
      Move(in := "Unit1.Em1.ControlNodes".cmRadiusMeasure.monitoring.Diameter, out1 => "Unit1.EmNodes".emRelations.em1.monitoring.UserDefine.diameter)
   END_RUNG
   RUNG wire#w1
      S_Move(in := "Unit1.Em1.HmiInterface".cmBobinID.monitoring.ResultData.datRead1, out => "Unit1.EmNodes".emRelations.em1.monitoring.UserDefine.bobinID)
   END_RUNG
   RUNG wire#w1
      Move(in := "BA010AZCRSP503.01", out1 => "Unit1.EmNodes".emRelations.em1.monitoring.UserDefine.RadiusAnaloge)
   END_RUNG
   // the same network as SCL:
   "Unit1.EmNodes".emRelations.em1.monitoring.UserDefine.winderDirectionChange := #TRUE AND "Unit1.Em1.HmiInterface".cmWinderDirectionChange;
   IF #TRUE THEN
       "Unit1.EmNodes".emRelations.em1.monitoring.UserDefine.radius := "Unit1.Em1.ControlNodes".cmRadiusMeasure.monitoring.Radius;
       "Unit1.EmNodes".emRelations.em1.monitoring.UserDefine.diameter := "Unit1.Em1.ControlNodes".cmRadiusMeasure.monitoring.Diameter;
       "Unit1.EmNodes".emRelations.em1.monitoring.UserDefine.bobinID := "Unit1.Em1.HmiInterface".cmBobinID.monitoring.ResultData.datRead1;
       "Unit1.EmNodes".emRelations.em1.monitoring.UserDefine.RadiusAnaloge := "BA010AZCRSP503.01";
   END_IF;
END_REGION

REGION Network 106: SyncMotion Configuration
   RUNG wire#powerrail
      Move(in := "Unit1.Em1.Config".axis[1], out1 => "Unit1.MotionNodes".PLCToMotion.TechnologyObject.Axis.UnwinderRight)
      Contact( #emFeedback.isLinked )
      Coil( "Unit1.MotionNodes".PLCToMotion.Parameter.Dancer.UnwinderRightUse )
   END_RUNG
   // the same network as SCL:
   "Unit1.MotionNodes".PLCToMotion.TechnologyObject.Axis.UnwinderRight := "Unit1.Em1.Config".axis[1];
   "Unit1.MotionNodes".PLCToMotion.Parameter.Dancer.UnwinderRightUse := #emFeedback.isLinked;
END_REGION

REGION Network 107: Em Nodes Brake Test
   RUNG wire#powerrail
      Contact( "Unit1.Em1.ControlNodes".cm.brakeTest.unwinder.monitoring.busy )
      Coil( "Unit1.EmNodes".allBrakeTest.monitoring.emStatus.busy[1] )
   END_RUNG
   RUNG wire#powerrail
      Contact( "Unit1.Em1.ControlNodes".cm.brakeTest.unwinder.monitoring.complete )
      Coil( "Unit1.EmNodes".allBrakeTest.monitoring.emStatus.complete[1] )
   END_RUNG
   RUNG wire#powerrail
      Contact( "Unit1.Em1.ControlNodes".cm.brakeTest.unwinder.monitoring.ready )
      Coil( "Unit1.EmNodes".allBrakeTest.monitoring.emStatus.axisEnabled[1] )
   END_RUNG
   // the same network as SCL:
   "Unit1.EmNodes".allBrakeTest.monitoring.emStatus.busy[1] := "Unit1.Em1.ControlNodes".cm.brakeTest.unwinder.monitoring.busy;
   "Unit1.EmNodes".allBrakeTest.monitoring.emStatus.complete[1] := "Unit1.Em1.ControlNodes".cm.brakeTest.unwinder.monitoring.complete;
   "Unit1.EmNodes".allBrakeTest.monitoring.emStatus.axisEnabled[1] := "Unit1.Em1.ControlNodes".cm.brakeTest.unwinder.monitoring.ready;
END_REGION
END_FUNCTION_BLOCK
